TYPE "ESD_SET"
VERSION : 0.1
   STRUCT
      Delay_time : Time;   // Задержка включения противоаварийной защиты
      Limit : Real;   // Предел противоаварийной защиты (если используется)
      Hyst : Real;   // Гистерезис срабатывания (если используется)
      TEST : Bool;   // Тест противоавариной защиты
      DEBLOCK : Bool;   // Деблокировка (деактивация) противоавариной защиты
   END_STRUCT;

END_TYPE

